TYPE ST_Enclosure_get :
STRUCT
	climate				: REFERENCE TO ST_EnclosureClimate_Get;
	doors				: REFERENCE TO ST_DoorsNLocks_events;
	ledstrip			: REFERENCE TO ST_Ledstrip_events;
END_STRUCT
END_TYPE

(* stored: Version 1.1.0.1, ProductVersion 3.1.4024.12
   DUT ST_Enclosure_get: Id {a884b94b-5278-45e4-8e11-5ffcd334137c} *)
